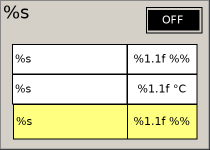
VISUALIZATION VISU_CHAUFF  // 210x150
VAR_IN_OUT
	m_Input_ELMT_CHAUFF:	BLOCK_ELMT_CHAUFF;
END_VAR
    Rectangle (0,0 210x150), "%s", text list: 'TextList_Chauffage', text index: 0
    RoundedRectangle (12,44 115x30), "%s", text list: 'TextList_Chauffage', text index: 1
    RoundedRectangle (127,44 70x30), "%1.1f %%", text variable: m_Input_ELMT_CHAUFF.OUT_QCH.Value
    RoundedRectangle (149,10 50x20), "ON", invisible if: NOT m_Input_ELMT_CHAUFF.OUT_MCH
    RoundedRectangle (148,10 50x20), "OFF", invisible if: m_Input_ELMT_CHAUFF.OUT_MCH
    RoundedRectangle (13,104 116x35), "%s", invisible if: NOT m_Input_ELMT_CHAUFF.PRM_Ctrl, input disabled if: NOT m_Input_ELMT_CHAUFF.MANUAL OR NOT PRG_USER.ACTU_USER.MAINTENANCE, text list: 'TextList_Chauffage', text index: 3
        OnMouseClick: toggle m_Input_ELMT_CHAUFF.PRM_Ctrl
    RoundedRectangle (127,104 70x35), "%1.1f °C", text variable: m_Input_ELMT_CHAUFF.PRM_Temperature, invisible if: NOT m_Input_ELMT_CHAUFF.PRM_Ctrl, input disabled if: NOT m_Input_ELMT_CHAUFF.MANUAL OR NOT PRG_USER.ACTU_USER.MAINTENANCE
        OnMouseClick: write the text variable via VisuDialogs.Numpad, min m_Input_ELMT_CHAUFF.CONF_TMIN, max m_Input_ELMT_CHAUFF.CONF_TMAX
    RoundedRectangle (127,74 70x30), "%1.1f °C", text variable: m_Input_ELMT_CHAUFF.IN_Temperature
    RoundedRectangle (12,74 115x30), "%s", text list: 'TextList_Chauffage', text index: 2
    RoundedRectangle (13,104 115x35), "%s", invisible if: m_Input_ELMT_CHAUFF.PRM_Ctrl, input disabled if: NOT m_Input_ELMT_CHAUFF.MANUAL OR NOT PRG_USER.ACTU_USER.MAINTENANCE, text list: 'TextList_Chauffage', text index: 4
        OnMouseClick: toggle m_Input_ELMT_CHAUFF.PRM_Ctrl
    RoundedRectangle (127,104 70x35), "%1.1f %%", text variable: m_Input_ELMT_CHAUFF.PRM_Power, invisible if: m_Input_ELMT_CHAUFF.PRM_Ctrl, input disabled if: NOT m_Input_ELMT_CHAUFF.MANUAL OR NOT PRG_USER.ACTU_USER.MAINTENANCE
        OnMouseClick: write the text variable via VisuDialogs.Numpad, min 0, max m_Input_ELMT_CHAUFF.CONF_PMAX
    Rectangle (146,7 56x26), invisible if: (NOT m_Input_ELMT_CHAUFF.AUTOR_Off_IHM AND NOT m_Input_ELMT_CHAUFF.AUTOR_On_IHM) OR NOT PRG_USER.ACTU_USER.MAINTENANCE, input disabled if: (NOT m_Input_ELMT_CHAUFF.AUTOR_Off_IHM AND NOT m_Input_ELMT_CHAUFF.AUTOR_On_IHM) OR NOT PRG_USER.ACTU_USER.MAINTENANCE
        tap m_Input_ELMT_CHAUFF.M_On
END_VISUALIZATION

(* stored: Version 1.1.0.1, ProductVersion 3.1.4024.10
   Visu VISU_CHAUFF: Id {747922e3-74c0-43fa-b7b5-c0c7b6387f70} *)
